PROGRAM PRG_ExtractStringManual
VAR
	fbExtractString		: FB_ExtractString;
	
	bExtractData		: BOOL;			(* set TRUE to remove prefix and suffix from strData *)
	nExtractChars		: UINT;			(* if suffix is blank, number of data chars to extract *)
	sPrefix				: T_MaxString;	(* prefix string *)
	sSuffix				: T_MaxString;	(* suffix string *)


	sDataString			: T_MaxString;	(* string to be searched *)

	bStringFound				: BOOL;			(* TRUE = sub-string with matching prefix/suffix found *)
	sExtractedString			: T_MaxString;	(* extracted data *)
	nExtractedStringPos			: UDINT;			(* start pos of extracted string in strString *)

	sResultString			: T_MaxString;	(* extracted data *)
END_VAR

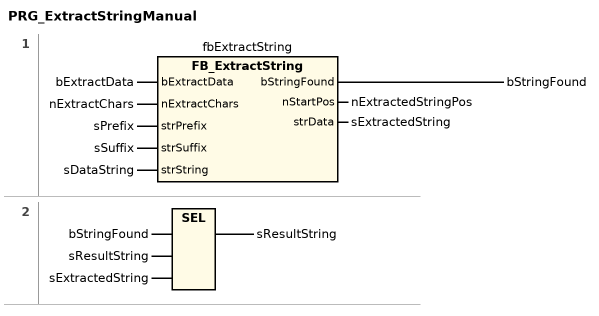
// NETWORK 1
fbExtractString(
    bExtractData := bExtractData,
    nExtractChars := nExtractChars,
    strPrefix := sPrefix,
    strSuffix := sSuffix,
    strString := sDataString,
    nStartPos => nExtractedStringPos,
    strData => sExtractedString); // FB_ExtractString
bStringFound := fbExtractString.bStringFound;

// NETWORK 2
sResultString := SEL(bStringFound, sResultString, sExtractedString);

END_PROGRAM

(* stored: Version 1.1.0.1
   POU PRG_ExtractStringManual: Id {de92ac7f-9b93-4f27-9238-6b20c8cc3656}, SpecialFunc None *)
